METHOD M_ManualAllocateHoming
VAR_INPUT
END_VAR
//fbAllocateArea.fbAllocateHome.xExecute := Service_Handshake.AllocationRegionHome.HandShake.Execute;
IF Service_Handshake.AllocationRegionHome.HandShake.Execute THEN
	fbAllocateArea.M_StartHoming();
END_IF
Service_Handshake.AllocationRegionHome.HandShake.Busy := fbAllocateArea.fbAllocateHome.xBusy;
Service_Handshake.AllocationRegionHome.HandShake.Done := fbAllocateArea.fbAllocateHome.xDone;
Service_Handshake.AllocationRegionHome.HandShake.Error := fbAllocateArea.fbAllocateHome.xError;
IF  NOT Service_Handshake.AllocationRegionHome.HandShake.Execute THEN
	fbAllocateArea.M_StopHoming();
END_IF

Service_Handshake.AllocationRegionHome.Homed := fbAllocateArea.Homed;
END_METHOD

METHOD PRIVATE M_ManualMachineHome
VAR_INPUT
END_VAR
IF Service_Handshake.MachineHome.HandShake.Execute THEN
	M_StartHoming();
END_IF
Service_Handshake.MachineHome.HandShake.Busy := fbMachineHoming.xBusy;
Service_Handshake.MachineHome.HandShake.Done  := fbMachineHoming.xDone;
Service_Handshake.MachineHome.HandShake.Error := fbMachineHoming.xError;
IF NOT Service_Handshake.MachineHome.HandShake.Execute THEN
	M_StopHoming();
END_IF

Service_Handshake.MachineHome.Homed := MachineHomed;
END_METHOD

METHOD M_ManualShippingHoming 
VAR_INPUT
END_VAR
//fbStorageArea.fbStoragehoming.xExecute := Service_Handshake.StorageRegionHome.HandShake.Execute;
IF Service_Handshake.FGARegionHome.HandShake.Execute THEN
	fbShippingArea.M_StartHoming();
END_IF
Service_Handshake.FGARegionHome.HandShake.Busy := fbShippingArea.fbshippinghoming.xBusy;
Service_Handshake.FGARegionHome.HandShake.Done := fbShippingArea.fbshippinghoming.xDone;
Service_Handshake.FGARegionHome.HandShake.Error := fbShippingArea.fbshippinghoming.xError;
IF NOT Service_Handshake.FGARegionHome.HandShake.Execute  THEN
	fbShippingArea.M_StopHoming();
END_IF

Service_Handshake.FGARegionHome.Homed := fbShippingArea.Homed;
END_METHOD

METHOD M_ManualStorageHoming
VAR_INPUT
END_VAR
//fbStorageArea.fbStoragehoming.xExecute := Service_Handshake.StorageRegionHome.HandShake.Execute;
IF Service_Handshake.StorageRegionHome.HandShake.Execute THEN
	fbStorageArea.M_StartHoming();
END_IF
Service_Handshake.StorageRegionHome.HandShake.Busy := fbStorageArea.fbStoragehoming.xBusy;
Service_Handshake.StorageRegionHome.HandShake.Done := fbStorageArea.fbStoragehoming.xDone;
Service_Handshake.StorageRegionHome.HandShake.Error := fbStorageArea.fbStoragehoming.xError;
IF  NOT Service_Handshake.StorageRegionHome.HandShake.Execute THEN
	fbStorageArea.M_StopHoming();
END_IF

Service_Handshake.StorageRegionHome.Homed := fbStorageArea.Homed;
END_METHOD

METHOD M_Resetting
VAR
	CylinderIndex : INT;
	MotorIndex : INT;
END_VAR
FOR CylinderIndex := 1 TO 53 DO
	fbAllocateArea.M_TransCVCameraPress_ManualMode();
    Cylinder.arCylinder[CylinderIndex].xEnable := TRUE;
	CylinderManualCtrl[CylinderIndex].Cylinder REF= Cylinder.arCylinder[CylinderIndex];
END_FOR

FOR CylinderIndex := 1 TO 53 DO
    Cylinder.arCylinder[CylinderIndex].EnableSimulation := EnableSimulation;
END_FOR

FOR MotorIndex := 1 TO 26 DO
    Motor.arMotor[MotorIndex].xEnable := TRUE;
	MotorManualCtrl[MotorIndex].Motor REF= Motor.arMotor[MotorIndex];
END_FOR

// Reference 
ReferenceHMI();
RefStorageService();
RefAllocateService();
RefShippingService();

// State control
GVL_Machine.PackTags[UnitNo.Allocate].Command.CntrlCmd := ePMLCommand_Reset;
GVL_Machine.PackTags[UnitNo.Storage].Command.CntrlCmd := ePMLCommand_Reset;
GVL_Machine.PackTags[UnitNo.Shipping].Command.CntrlCmd := ePMLCommand_Reset;
arAxisCtrl_gb[AxisNo.RoundBelt].Admin.PositionType := E_PositionType.Modulo;
arAxisCtrl_gb[AxisNo.TurnTable].Admin.PositionType := E_PositionType.Modulo;

CASE eModeCurrent OF
    E_UnitMode.Manual:
        IF GVL_Machine.PackTags[UnitNo.Allocate].Status.StateCurrent = ePMLState_Idle AND
            GVL_Machine.PackTags[UnitNo.Storage].Status.StateCurrent = ePMLState_Idle AND
            GVL_Machine.PackTags[UnitNo.Shipping].Status.StateCurrent = ePMLState_Idle //
			 THEN
            M_StateComplete();
        END_IF
		IF ErrorTableInitDone THEN
			M_General_AlarmRegister();
		END_IF
    E_UnitMode.Auto:
        IF GVL_Machine.PackTags[UnitNo.Allocate].Status.StateCurrent = ePMLState_Idle AND
            GVL_Machine.PackTags[UnitNo.Storage].Status.StateCurrent = ePMLState_Idle AND
            GVL_Machine.PackTags[UnitNo.Shipping].Status.StateCurrent = ePMLState_Idle //AND
             THEN
            M_StateComplete();
        END_IF
		IF ErrorTableInitDone THEN
			M_General_AlarmRegister();
		END_IF
END_CASE
END_METHOD

METHOD M_StartHoming
VAR_INPUT
END_VAR
fbMachineHoming.xExecute := TRUE;
END_METHOD

METHOD M_Starting
// State control
GVL_Machine.PackTags[UnitNo.Allocate].Command.CntrlCmd := ePMLCommand_Start;
GVL_Machine.PackTags[UnitNo.Storage].Command.CntrlCmd := ePMLCommand_Start;
GVL_Machine.PackTags[UnitNo.Shipping].Command.CntrlCmd := ePMLCommand_Start;

CASE eModeCurrent OF
    E_UnitMode.Manual, E_UnitMode.Auto:
        IF GVL_Machine.PackTags[UnitNo.Allocate].Status.StateCurrent = ePMLState_Execute AND
            GVL_Machine.PackTags[UnitNo.Allocate].Status.StateCurrent = ePMLState_Execute AND
            GVL_Machine.PackTags[UnitNo.Allocate].Status.StateCurrent = ePMLState_Execute THEN
            M_StateComplete();
        END_IF
END_CASE
END_METHOD

METHOD M_StopHoming
VAR_INPUT
END_VAR
fbMachineHoming.xExecute := FALSE;
END_METHOD

METHOD M_Stopped
VAR
	CylinderIndex : INT;
	MotorIndex : INT;
	ServoIndex : INT;
END_VAR
FOR ServoIndex := 1 TO 7 DO
	IF arAxisCtrl_gb[ServoIndex].Admin.Axis.Status.Error THEN
		arAxisCtrl_gb[ServoIndex].Admin.ClearError := FALSE;
	END_IF
END_FOR

IF eModeCurrent = E_UnitMode.Auto THEN
	GVL_Machine.PackTags[UnitNo.Storage].Command.UnitMode := E_UnitMode.Auto;
	GVL_Machine.PackTags[UnitNo.Allocate].Command.UnitMode := E_UnitMode.Auto;
	GVL_Machine.PackTags[UnitNo.Shipping].Command.UnitMode := E_UnitMode.Auto;
ELSIF eModeCurrent = E_UnitMode.Manual THEN
	GVL_Machine.PackTags[UnitNo.Storage].Command.UnitMode := E_UnitMode.Manual;
	GVL_Machine.PackTags[UnitNo.Allocate].Command.UnitMode := E_UnitMode.Manual;
	GVL_Machine.PackTags[UnitNo.Shipping].Command.UnitMode := E_UnitMode.Manual;
END_IF

CASE eModeCurrent OF
	E_UnitMode.Manual:
		IF GVL_Machine.PackTags[UnitNo.Allocate].Status.UnitModeCurrent = E_UnitMode.Manual AND 
			GVL_Machine.PackTags[UnitNo.Allocate].Status.StateCurrent = ePMLState_Stopped AND
			GVL_Machine.PackTags[UnitNo.Storage].Status.UnitModeCurrent = E_UnitMode.Manual AND 
			GVL_Machine.PackTags[UnitNo.Storage].Status.StateCurrent = ePMLState_Stopped AND
			GVL_Machine.PackTags[UnitNo.Shipping].Status.UnitModeCurrent = E_UnitMode.Manual AND 
			GVL_Machine.PackTags[UnitNo.Shipping].Status.StateCurrent = ePMLState_Stopped THEN
			M_StateComplete();
		END_IF
	E_UnitMode.Auto:
		IF GVL_Machine.PackTags[UnitNo.Allocate].Status.UnitModeCurrent = E_UnitMode.Auto AND 
			GVL_Machine.PackTags[UnitNo.Allocate].Status.StateCurrent = ePMLState_Stopped AND
			GVL_Machine.PackTags[UnitNo.Storage].Status.UnitModeCurrent = E_UnitMode.Auto AND 
			GVL_Machine.PackTags[UnitNo.Storage].Status.StateCurrent = ePMLState_Stopped AND
			GVL_Machine.PackTags[UnitNo.Shipping].Status.UnitModeCurrent = E_UnitMode.Auto AND 
			GVL_Machine.PackTags[UnitNo.Shipping].Status.StateCurrent = ePMLState_Stopped THEN
			M_StateComplete();
		END_IF
END_CASE
END_METHOD

METHOD M_Stopping
VAR
	CylinderIndex :INT;
	MotorIndex : INT;
END_VAR
CASE eModeCurrent OF
    E_UnitMode.Manual:
        GVL_Machine.PackTags[UnitNo.Allocate].Command.UnitMode := E_UnitMode.Manual;
        GVL_Machine.PackTags[UnitNo.Allocate].Command.CntrlCmd := ePMLCommand_Stop;
        GVL_Machine.PackTags[UnitNo.Storage].Command.UnitMode  := E_UnitMode.Manual;
        GVL_Machine.PackTags[UnitNo.Storage].Command.CntrlCmd  := ePMLCommand_Stop;
        GVL_Machine.PackTags[UnitNo.Shipping].Command.UnitMode := E_UnitMode.Manual;
        GVL_Machine.PackTags[UnitNo.Shipping].Command.CntrlCmd := ePMLCommand_Stop;
		FOR CylinderIndex := 1 TO 53 DO
			Cylinder.arCylinder[CylinderIndex].xEnable := FALSE;
		END_FOR
		FOR MotorIndex := 1 TO 26 DO
			Motor.arMotor[MotorIndex].xEnable := FALSE;
		END_FOR
		TableMove.xExecute := FALSE;
        IF GVL_Machine.PackTags[UnitNo.Allocate].Status.UnitModeCurrent = E_UnitMode.Manual AND
           GVL_Machine.PackTags[UnitNo.Allocate].Status.StateCurrent = ePMLState_Stopped AND
           GVL_Machine.PackTags[UnitNo.Storage].Status.UnitModeCurrent = E_UnitMode.Manual AND
           GVL_Machine.PackTags[UnitNo.Storage].Status.StateCurrent = ePMLState_Stopped AND
           GVL_Machine.PackTags[UnitNo.Shipping].Status.UnitModeCurrent = E_UnitMode.Manual AND
           GVL_Machine.PackTags[UnitNo.Shipping].Status.StateCurrent = ePMLState_Stopped AND NOT
		   TableMove.xError
            THEN
            M_StateComplete();
        END_IF
	E_UnitMode.Auto:
        GVL_Machine.PackTags[UnitNo.Allocate].Command.UnitMode := E_UnitMode.Auto;
        GVL_Machine.PackTags[UnitNo.Allocate].Command.CntrlCmd := ePMLCommand_Stop;
        GVL_Machine.PackTags[UnitNo.Storage].Command.UnitMode  := E_UnitMode.Auto;
        GVL_Machine.PackTags[UnitNo.Storage].Command.CntrlCmd  := ePMLCommand_Stop;
        GVL_Machine.PackTags[UnitNo.Shipping].Command.UnitMode := E_UnitMode.Auto;
        GVL_Machine.PackTags[UnitNo.Shipping].Command.CntrlCmd := ePMLCommand_Stop;
		FOR CylinderIndex := 1 TO 53 DO
			Cylinder.arCylinder[CylinderIndex].xEnable := FALSE;
		END_FOR
		FOR MotorIndex := 1 TO 26 DO
			Motor.arMotor[MotorIndex].xEnable := FALSE;
		END_FOR
		TableMove.xExecute := FALSE;
        IF GVL_Machine.PackTags[UnitNo.Allocate].Status.UnitModeCurrent = E_UnitMode.Auto AND
           GVL_Machine.PackTags[UnitNo.Allocate].Status.StateCurrent = ePMLState_Stopped AND
           GVL_Machine.PackTags[UnitNo.Storage].Status.UnitModeCurrent = E_UnitMode.Auto AND
           GVL_Machine.PackTags[UnitNo.Storage].Status.StateCurrent = ePMLState_Stopped AND
           GVL_Machine.PackTags[UnitNo.Shipping].Status.UnitModeCurrent = E_UnitMode.Auto AND
           GVL_Machine.PackTags[UnitNo.Shipping].Status.StateCurrent = ePMLState_Stopped AND NOT
		   TableMove.xError
            THEN
            M_StateComplete();
        END_IF
END_CASE
END_METHOD

METHOD PRIVATE M_StroageRobotSafeCheck : BOOL
VAR_INPUT
END_VAR
IF FanucRobot.List.StorageRobot._DI12.BzoneWaitAllow THEN
	IF NOT arAxisCtrl_gb[AxisNo.RoundBelt].Admin.Axis.Status.Moving
	    AND NOT fbAllocateArea.RoundBeltControl.xBusy
		AND NOT fbAllocateArea.RoundBeltControl.xError
		AND NOT fbAllocateArea.RoundBeltControl.xDone THEN
			FanucRobot.List.StorageRobot.Bzone_AllowWork := TRUE;
	END_IF
END_IF

IF NOT FanucRobot.List.StorageRobot._DI12.BzoneInWork 
	AND NOT FanucRobot.List.StorageRobot._DI12.BzoneWaitAllow THEN
	FanucRobot.List.StorageRobot.Bzone_AllowWork := FALSE	;
END_IF
END_METHOD

METHOD M_Suspended
M_StateComplete();
END_METHOD

METHOD M_Suspending
M_StateComplete();
END_METHOD

METHOD M_Undefined
CASE eModeCurrent OF
    E_UnitMode.Undefined:
		PackTag.Command.UnitMode := E_UnitMode.Manual;
		PackTag.Command.CntrlCmd := ePMLCommand_Abort;
		M_StateComplete();
END_CASE
END_METHOD

METHOD M_Unholding
M_StateComplete();
END_METHOD

METHOD M_Unsuspending
END_METHOD

METHOD PRIVATE RefAllocateService
VAR_INPUT
END_VAR
AllocateService.AllocateMoveStructure 				REF= Service_Handshake.AllocateMoveStructure;
AllocateService.AllocateCircleMove 					REF= Service_Handshake.AllocateCircleMove;
AllocateService.TurnTableMove 						REF= Service_Handshake.TurnTableMove;

// Allocating
AllocateService.AutoMode_AllocateBatchMode 			REF= Service_Handshake.AutoMode_AllocateBatchMode;
AllocateService.AutoMode_SimpleAllocation_Batch 	REF= Service_Handshake.AutoMode_SimpleAllocation_Batch;
AllocateService.AutoMode_AllocateBatchMode_Reverse  REF= Service_Handshake.AutoMode_AllocateBatchMode_Reverse;

//OutRobot
AllocateService.AutoMode_RareBoxMove 				REF= Service_Handshake.AutoMode_RareBoxMove;
AllocateService.AutoMode_EmptyBoxMove 				REF= Service_Handshake.AutoMode_EmptyBoxMove;
AllocateService.AutoMode_BoxMoveReverse 			REF= Service_Handshake.AutoMode_BoxMoveReverse;

//TransCV camera 
AllocateService.AutoMode_SameSizeCVCamera 			REF= Service_Handshake.AutoMode_SameSizeCVCamera;
AllocateService.AutoMode_DifferentCVCamera 			REF= Service_Handshake.AutoMode_DifferentCVCamera;

//AllocateArea Home
AllocateService.AllocateRegionHome					REF= Service_Handshake.AllocationRegionHome;

// Pullout 
AllocateService.AutoMode_PullOutConveyor 			REF= Service_Handshake.AutoMode_PullOutConveyor;

//AutoModeUse*-------自動模式圓帶單動
   AllocateService.AutoMode_AllocateCircleMove 		 REF= Service_Handshake.AutoMode_AllocateCircleMove;

 //AutoModeUse*-------圓盤移動
    AllocateService.AutoMode_TurnTableMOve  		REF= Service_Handshake.AutoMode_TurnTableMOve;
	
//Allocate robot move
AllocateService.AllocateRobotNeedlingMove 			REF= Service_Handshake.AllocationRobotNeedlingMove;
END_METHOD

METHOD PRIVATE ReferenceHMI
VAR_INPUT
END_VAR
Service_Handshake.AllocateMoveStructure REF= GVL_ADS.AllocateMoveStructure;
Service_Handshake.AllocateMoveStructure_Reverse REF= GVL_ADS.AllocateMoveStructure_Reverse;
Service_Handshake.EmptyRobotToTurnTableMove REF= GVL_ADS.EmptyRobotToTurnTableMove;
Service_Handshake.AllocateCircleMove REF= GVL_ADS.AllocateCircleMove;
Service_Handshake.TurnTableMove REF= GVL_ADS.TurnTableMove;
//Service_Handshake.AxesControl REF= GVL_ADS.AxesControl;
Service_Handshake.MachineReset REF= GVL_ADS.MachineReset;
Service_Handshake.RareFullBoxPush REF= GVL_ADS.RareFullBoxPush;
Service_Handshake.AutoMode_AllocateCircleMove REF= GVL_ADS.AutoMode_AllocateCircleMove;
Service_Handshake.AutoMode_RobotWarehouseMove REF= GVL_ADS.AutoMode_RobotWarehouseMove;
Service_Handshake.AutoMode_RobotAbsMove REF= GVL_ADS.AutoMode_RobotAbsMove;
Service_Handshake.AutoMode_EmptyBoxMove REF= GVL_ADS.AutoMode_EmptyBoxMove;
Service_Handshake.AutoMode_TurnTableMOve REF= GVL_ADS.AutoMode_TurnTableMOve;
Service_Handshake.AutoMode_AllocateMove REF= GVL_ADS.AutoMode_AllocateMove;
Service_Handshake.AutoMode_AllocateMove_Reverse REF= GVL_ADS.AutoMode_AllocateMove_Reverse;
Service_Handshake.AutoMode_AllocateBatchMode REF= GVL_ADS.AutoMode_AllocateBatchMode;
Service_Handshake.AutoMode_AllocateBatchMode_Reverse REF= GVL_ADS.AutoMode_AllocateBatchMode_Reverse;
Service_Handshake.AutoMode_SimpleAllocation_Batch REF= GVL_ADS.AutoMode_SimpleAllocation_Batch;
Service_Handshake.AutoMode_RareBoxMove REF= GVL_ADS.AutoMode_RareBoxMove;
Service_Handshake.AutoMode_OutBoxMove REF= GVL_ADS.AutoMode_OutBoxMove;
Service_Handshake.AutoMode_BoxMoveReverse REF= GVL_ADS.AutoMode_BoxMoveReverse;
Service_Handshake.AutoMode_WarehouseMove REF= GVL_ADS.AutoMode_WarehouseMove;
Service_Handshake.AutoMode_ErrorHandle REF= GVL_ADS.AutoMode_ErrorHandle;
Service_Handshake.AlarmAllocation REF= GVL_ADS.AlarmAllocation;
Service_Handshake.AutoMode_MoveConveyorJob REF= GVL_ADS.AutoMode_MoveConveyorJob;
Service_Handshake.AutoMode_WarehouseMotoWithRobotMove REF= GVL_ADS.AutoMode_WarehouseMotoWithRobotMove;
Service_Handshake.AutoMode_SimpleAllocate REF= GVL_ADS.AutoMode_SimpleAllocate;
Service_Handshake.AutoMode_PullOutConveyor REF= GVL_ADS.AutoMode_PullOutConveyor;
Service_Handshake.AutoMode_AddBoxes REF= GVL_ADS.AutoMode_AddBoxes;
Service_Handshake.MachineHome REF= GVL_ADS.MachineHome;
Service_Handshake.StorageRegionHome REF= GVL_ADS.StorageRegionHome;
Service_Handshake.AllocationRegionHome REF= GVL_ADS.AllocationRegionHome;
Service_Handshake.FGARegionHome REF= GVL_ADS.FGARegionHome;
Service_Handshake.StorageRegionMode REF= GVL_ADS.StorageRegionMode;
Service_Handshake.AllocationRegion REF= GVL_ADS.AllocationRegion;
Service_Handshake.FGARegionMode REF= GVL_ADS.FGARegionMode;
Service_Handshake.MachineMode REF= GVL_ADS.MachineMode;
Service_Handshake.OpPannel_Status REF= GVL_ADS.OpPannel_Status;
Service_Handshake.OpPannel_Ctrl REF= GVL_ADS.OpPannel_Ctrl;
Service_Handshake.FanucRobot_General REF= GVL_ADS.FanucRobot_General;
Service_Handshake.AutoMode_FeedInEmptyBoxWithRobot REF= GVL_ADS.AutoMode_FeedInEmptyBoxWithRobot;
Service_Handshake.AutoMode_ReloadRoundBeltBoxWithRobot REF= GVL_ADS.AutoMode_ReloadRoundBeltBoxWithRobot;
Service_Handshake.AutoMode_UpperFeedInConveyor REF= GVL_ADS.AutoMode_UpperFeedInConveyor;
//Service_Handshake.MachineState REF= GVL_ADS.MachineState;
Service_Handshake.AutoMode_RobotRegionMove_FeedInConveyor REF= GVL_ADS.AutoMode_RobotRegionMove_FeedInConveyor;
Service_Handshake.AutoMode_RobotRegionMove_AllocatedConveyor REF= GVL_ADS.AutoMode_RobotRegionMove_AllocatedConveyor;
Service_Handshake.AutoMode_RobotRegionMove_PullOutConveyor REF= GVL_ADS.AutoMode_RobotRegionMove_PullOutConveyor;
Service_Handshake.AutoMode_RobotRegionMove_BufferArea REF= GVL_ADS.AutoMode_RobotRegionMove_BufferArea;
Service_Handshake.AutoMode_RobotRegionMove_RoundBelt REF= GVL_ADS.AutoMode_RobotRegionMove_RoundBelt;
Service_Handshake.AutoMode_ShippingRobot_Left REF= GVL_ADS.AutoMode_ShippingRobot_Left;
Service_Handshake.AutoMode_ShippingRobot_Right REF= GVL_ADS.AutoMode_ShippingRobot_Right;
Service_Handshake.AutoMode_ShippingRobot_TransmitCVEnd REF= GVL_ADS.AutoMode_ShippingRobot_TransmitCVEnd;
Service_Handshake.AutoMode_SameSizeCVCamera REF= GVL_ADS.AutoMode_SameSizeCVCamera;
Service_Handshake.AutoMode_DifferentCVCamera REF= GVL_ADS.AutoMode_DifferentCVCamera;

Service_Handshake.AllocationRobotNeedlingMove REF= GVL_ADS.AllocationRobotNeedlingMove;
END_METHOD

METHOD RefShippingService
VAR_INPUT
END_VAR
ShippingService.AutoMode_ShippingRobot_Left REF= Service_Handshake.AutoMode_ShippingRobot_Left;
ShippingService.AutoMode_ShippingRobot_Right REF= Service_Handshake.AutoMode_ShippingRobot_Right;
ShippingService.AutoMode_ShippingRobot_TransmitCVEnd REF= Service_Handshake.AutoMode_ShippingRobot_TransmitCVEnd;
END_METHOD

METHOD PRIVATE RefStorageService
VAR_INPUT
END_VAR
StorageService.AutoMode_ReloadRoundBeltBoxWithRobot	REF= Service_Handshake.AutoMode_ReloadRoundBeltBoxWithRobot;
StorageService.AutoMode_FeedInEmptyBoxWithRobot REF= Service_Handshake.AutoMode_FeedInEmptyBoxWithRobot;
StorageService.AutoMode_RobotRegionMove_FeedInConveyor REF= Service_Handshake.AutoMode_RobotRegionMove_FeedInConveyor;
StorageService.AutoMode_RobotRegionMove_AllocatedConveyor REF= Service_Handshake.AutoMode_RobotRegionMove_AllocatedConveyor;
StorageService.AutoMode_RobotRegionMove_PullOutConveyor REF= Service_Handshake.AutoMode_RobotRegionMove_PullOutConveyor;
StorageService.AutoMode_RobotRegionMove_BufferArea REF= Service_Handshake.AutoMode_RobotRegionMove_BufferArea;
StorageService.AutoMode_RobotRegionMove_RoundBelt REF= Service_Handshake.AutoMode_RobotRegionMove_RoundBelt;
StorageService.AutoMode_UpperFeedInConveyor REF=  Service_Handshake.AutoMode_UpperFeedInConveyor;
StorageService.AutoMode_AddBoxes REF= Service_Handshake.AutoMode_AddBoxes;
StorageService.AutoMode_PullOutConveyor REF= Service_Handshake.AutoMode_PullOutConveyor;
StorageService.AutoMode_RobotAbsMove REF=  Service_Handshake.AutoMode_RobotAbsMove;
StorageService.AutoMode_WarehouseMotoWithRobotMove REF= Service_Handshake.AutoMode_WarehouseMotoWithRobotMove;
END_METHOD

END_FUNCTION_BLOCK

(* stored: Version 1.1.0.1, ProductVersion 3.1.4024.13
   POU FB_MachineControl: Id {e3b1bb4d-882f-4a96-a73d-3761a8a6d18d}, SpecialFunc None
   Folder Privite: Id {d682bfe9-5092-4ebc-ab4e-f307c30573aa}
   Folder Auto: Id {78745a11-46b7-4748-8552-0bd2d3b5d4a6}
   Folder HalfAuto: Id {99264d16-3d80-4746-9baf-d0c3138ca219}
   Folder HMI_Handshake: Id {bf445d25-6f86-4a62-a9d1-6ae38a86fa4a}
   Folder Manual: Id {25c13a10-8a56-4119-be12-75ef3638d999}
   Folder Service: Id {97187d91-1374-40f7-a3bd-68a8e6324174}
   Folder States: Id {6cde1021-8eff-4f8d-b6d5-827659856462}
   Action A00_BaseUnits: Id {c7c8760f-56d1-4aff-9f21-aabead4ce11d}
   Action A01_Cylinder: Id {03239220-aa5d-45c0-a759-6c4a9a88feea}
   Action A02_Motor: Id {5b2083a4-a76e-49c8-96ac-9e1562db4135}
   Action A03_FanucRobot: Id {bb200e91-8356-4c56-8d68-26872b17f60a}
   Action A04_OpPannel: Id {bd9ff175-ff19-4976-8958-fe3c79e5468c}
   Action A05_Light: Id {6a000875-27c0-4eef-9aa2-70b57063df14}
   Action A10_ErrorHandler: Id {6e15a011-548e-48fd-a150-b888d730dc27}
   Method M_Aborted: Id {07590437-cdc2-4926-8c27-767ace7419e7}
   Method M_Aborting: Id {8655fba0-b509-44e8-9ec4-a94584b04c87}
   Method M_Auto_Axes: Id {0e064b18-95a3-46b5-ad34-93887c3bb466}
   Method M_Clearing: Id {f7b9b0cb-7b5c-4dcd-9a94-060df5e92c19}
   Method M_ClearOutput: Id {873f93ff-c409-4eca-ad17-a178722c91ec}
   Method M_Complete: Id {d708bc1d-909d-41c5-938c-4fa8a3d42458}
   Method M_Completing: Id {4fc04777-9f54-4a57-badb-2e3830f1ee6b}
   Method M_Execute: Id {560a1df4-f108-4f5f-9158-749967ef08a7}
   Method M_General_AlarmRegister: Id {3ef4b090-7ef0-4623-ae15-9f802c71cf11}
   Method M_GetCylinderError: Id {10e6797e-0ae1-48b1-a1ef-c777dcfd9688}
   Method M_HalfAuto_TableMove: Id {83a60461-797f-41e8-a820-71275e852ddf}
   Method M_Held: Id {420ce41a-bf89-41b1-a8c7-0faea8e9cb0a}
   Method M_Holding: Id {79dc20ca-afb0-4f06-82f1-0ce6b40186e7}
   Method M_Idle: Id {6f8ed9f5-2f19-457b-9f22-1fe1866c0063}
   Method M_MachineHoming: Id {6cd39fea-2cd0-47af-b417-30a765567e6c}
   Method M_Manual_Axes: Id {1febef1b-de19-40fb-b84d-01cddba8dd63}
   Method M_Manual_Cylinder: Id {cbaf563d-59fe-4de2-b76e-928a4c9b9648}
   Method M_Manual_Motor: Id {075b07e5-6665-4c9d-aa5b-ce8d0fed42d1}
   Method M_ManualAllocateHoming: Id {f1049744-2f7f-4913-b4df-5d6efedeb6f8}
   Method M_ManualMachineHome: Id {0386eb3f-5698-4a4c-acd8-c29dc86a27dd}
   Method M_ManualShippingHoming: Id {a052a37b-f4cf-460d-8831-592148b0b1ab}
   Method M_ManualStorageHoming: Id {59800549-b7c8-4847-b683-c0e8fab8b4be}
   Method M_Resetting: Id {8a313413-a9db-4d95-862c-f955afe04d5f}
   Method M_StartHoming: Id {1cfc2ec4-8978-47d1-a618-ea9ffb09495f}
   Method M_Starting: Id {6b0ffb98-6d92-4abc-97da-1afb9c25afa1}
   Method M_StopHoming: Id {bda1385e-b549-4a20-9f6b-8090d194cc8f}
   Method M_Stopped: Id {cd99af5a-54e9-48b9-8604-5ab42447d75f}
   Method M_Stopping: Id {13bedb0a-797e-46e7-b980-19fbd19b81d3}
   Method M_StroageRobotSafeCheck: Id {47e1cb93-7251-463c-9d1e-e7a9c6d5d136}
   Method M_Suspended: Id {7615c7fb-fc07-40e0-962d-50cdae246718}
   Method M_Suspending: Id {08514eda-eb99-46b5-a548-80121dc964e9}
   Method M_Undefined: Id {ebe3ecb5-5439-46a1-8ace-e8495c074189}
   Method M_Unholding: Id {64e7d9e3-bbb6-44d4-85b6-aa16778f4162}
   Method M_Unsuspending: Id {90314e7c-5afc-42b9-bfd4-0393ed17b222}
   Method RefAllocateService: Id {7e2d0ea7-efb8-45f5-8e87-93fdf1e313ed}
   Method ReferenceHMI: Id {f6889bed-a428-4faa-8d67-c5add5d80ffa}
   Method RefShippingService: Id {dcbecbba-f47d-4888-8ded-1da584981d0d}
   Method RefStorageService: Id {1a766cf2-e5ed-4657-8a78-f09a69ade618} *)
